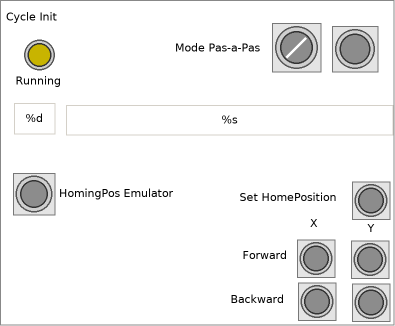
VISUALIZATION VisuInit  // 395x326
    Lamp1 (21,37 37x36), variable: fbCycleInit.xBusy, style: Lamp-Lamp1-Yellow
    Label (3,2 137x30), "Cycle Init"
    Label (9,66 59x30), "Running"
    Textfield (66,105 327x30), "%s", text variable: fbCycleInit.fbEtape.sMess
    Textfield (14,103 41x31), "%d", text variable: fbCycleInit.iEtape
    RotarySwitch (272,22 49x51), variable: stParam.stStatus.xModePasAPas, behaviour: TOGGLE, style: Switch-RotarySwitch-Gray
    Label (152,33 111x30), "Mode Pas-a-Pas"
    PushSwitch (13,173 42x42), tooltip "Do next step if Pas-a-Pas is enabled", variable: stIO.stIn.xHomingPosReached, invisible if: stParam.stStatus.xHomingDone, behaviour: TAP, style: Switch-PushSwitch-Gray
    Label (56,180 139x27), "HomingPos Emulator", invisible if: stParam.stStatus.xHomingDone
    PushSwitch (332,25 46x48), tooltip "Do next step if Pas-a-Pas is enabled", variable: fbBtn.xNextPas, behaviour: TAP, style: Switch-PushSwitch-Gray
    Group (191,179 199x145)
        Label (2,62 97x29), "Forward", invisible if: fbCycleInit.iEtape<>500
        Label (0,106 96x29), "Backward", invisible if: fbCycleInit.iEtape<>500
        Group (46,0 153x145)
            PushSwitch (115,0 38x43), variable: stIO.stIn.xSetHomePos, invisible if: fbCycleInit.iEtape<>500, behaviour: TAP, style: Switch-PushSwitch-Gray
            Label (0,4 102x29), "Set HomePosition", invisible if: fbCycleInit.iEtape<>500
            PushSwitch (60,58 38x43), variable: stIO.stIn.xJogXForward, invisible if: fbCycleInit.iEtape<>500, behaviour: TAP, style: Switch-PushSwitch-Gray
            PushSwitch (115,102 38x43), variable: stIO.stIn.xJogYBackward, invisible if: fbCycleInit.iEtape<>500, behaviour: TAP, style: Switch-PushSwitch-Gray
            PushSwitch (114,59 38x43), variable: stIO.stIn.xJogYForward, invisible if: fbCycleInit.iEtape<>500, behaviour: TAP, style: Switch-PushSwitch-Gray
            PushSwitch (61,101 38x43), variable: stIO.stIn.xJogXBackward, invisible if: fbCycleInit.iEtape<>500, behaviour: TAP, style: Switch-PushSwitch-Gray
            Label (60,30 34x29), "X", invisible if: fbCycleInit.iEtape<>500
            Label (117,35 34x29), "Y", invisible if: fbCycleInit.iEtape<>500
END_VISUALIZATION

(* stored: Version 1.1.0.1, ProductVersion 3.1.4020.12
   Visu VisuInit: Id {328d1b28-1cb1-41b4-a0f7-1e71e74c49ed} *)
